{attribute 'GeneratedUsingTerminal: ATH2000-0250-0023'}
{attribute addProperty BoxType "ATH2000-0250-0023"}
{attribute addProperty Id "A_0015_ATH2040_5250_0022ATH2040_AE8CEE4614"}
{attribute addProperty CRC "3284314643"}
{attribute addProperty Size "14"}
TYPE A_0002_ATH2000_0250_0023_C3C2AA13 EXTENDS ATH2000_86175B41 :
STRUCT
	{attribute addProperty Name "A_0015_ATH2040_5250_0022"}
	{attribute addProperty PreviousPort "A_0002(ATH2000-0250-0023) : B"}
	A_0015_ATH2040_5250_0022 : ATH2040_AE8CEE46;
END_STRUCT
END_TYPE

(* stored: Version 1.2.0.0, ProductVersion 3.1.4024.9
   DUT A_0002_ATH2000_0250_0023_C3C2AA13: Id {741da131-fe47-480e-997a-dee285621620} *)
